(*			
	RafalOS
	Rafał Osajda		10.11.2025		TC 4024.66
	Główny blok konfiguracyjny MachineControl
*)
FUNCTION_BLOCK FB_MachineConfiguration EXTENDS FB_Base IMPLEMENTS ITF_MCConfiguration
VAR

END_VAR

(*			
	RafalOS
	Rafał Osajda		13.11.2025		TC 4024.66
	Metoda przeznaczona do dodawania elementów do FB_MachineControl
*)
METHOD AddElements : BOOL
VAR_INPUT
	itfMachineControl	: B_MachineControl.ITF_MCMachineControlConfigure;
END_VAR
END_METHOD

(*
	RafalOS
	Rafał Osajda		13.11.2025		TC 4024.66
	Dodanie samego siebie do systemu controli maszyny
*)
METHOD AddMachineCotrolToYourSelf : BOOL
VAR_INPUT
	itfMachineControl	: B_MachineControl.ITF_MCMachineControlConfigure;
END_VAR
END_METHOD

(*
	RafalOS
	Rafał Osajda		13.11.2025		TC 4024.66
	Dodanie modułu sterowania stanami i trybami do machinecontrol
*)
METHOD AddSaMCotrollerToMachineControl : BOOL
VAR_INPUT
	itfMachineControl	: B_MachineControl.ITF_MCMachineControlConfigure;
END_VAR
END_METHOD

(*			
	RafalOS
	Rafał Osajda		13.11.2025		TC 4024.66
	Zlinkowanie danych wspólnych do dodanych elementów
*)
METHOD LinkCommonDataToAddedElements : BOOL
VAR_INPUT
	itfMachineControl	: B_MachineControl.ITF_MCMachineControlConfigure;
END_VAR
END_METHOD

(*			
	RafalOS
	Rafał Osajda		13.11.2025		TC 4024.66
	Dodanie głównego komunikatora pomiędzy topelementami do topelementów
*)
METHOD LinkMassangerToaddedTopElements : BOOL
VAR_INPUT
	itfMachineControl	: B_MachineControl.ITF_MCMachineControlConfigure;
END_VAR
END_METHOD

(*			
	RafalOS
	Rafał Osajda		13.11.2025		TC 4024.66
	Podłączenie wsyzstkich zmiennych pochodzących od Programu safety 
*)
METHOD LinkSafetyToaddedElements : BOOL
VAR_INPUT
	itfMachineControl	: B_MachineControl.ITF_MCMachineControlConfigure;
END_VAR
END_METHOD

(*			
	RafalOS
	Rafał Osajda		13.11.2025		TC 4024.66
	Nadanie unikalnych kodów elementom w systemie
*)
METHOD SetCodeToAddedElements : BOOL
VAR_INPUT
	itfMachineControl	: B_MachineControl.ITF_MCMachineControlConfigure;
END_VAR
END_METHOD

(*			
	RafalOS
	Rafał Osajda		13.11.2025		TC 4024.66
	Nadaje unikalne ID zgłoszeniom dodanym do elementów w sesyemie
*)
METHOD SetIDEventsToAddedElements : BOOL
VAR_INPUT
	itfMachineControl	: B_MachineControl.ITF_MCMachineControlConfigure;
END_VAR
END_METHOD

(*			
	RafalOS
	Rafał Osajda		13.11.2025		TC 4024.66
	Dodanie wszystkim elementom w systemie unikalnego ID
*)
METHOD SetIDToAddedElements : BOOL
VAR_INPUT
	itfMachineControl	: B_MachineControl.ITF_MCMachineControlConfigure;
END_VAR
END_METHOD

END_FUNCTION_BLOCK

(* stored: Version 1.1.0.1, ProductVersion 3.1.4024.15
   POU FB_MachineConfiguration: Id {ee925a5b-f7fe-416e-8a33-e493e5327aae}, SpecialFunc None
   Method AddElements: Id {7b730765-41af-4c9b-9f6a-4c5a645abba8}
   Method AddMachineCotrolToYourSelf: Id {c8ed0d9d-f48c-476a-915b-a4eba002124b}
   Method AddSaMCotrollerToMachineControl: Id {01e4bd98-cea4-48b9-bac4-c2658d2eb279}
   Method LinkCommonDataToAddedElements: Id {ac0aabe4-15a4-490d-b3a0-5896b9031d05}
   Method LinkMassangerToaddedTopElements: Id {b7ca5c08-4047-434f-be66-47086ad067ba}
   Method LinkSafetyToaddedElements: Id {a7fb546a-9043-48d0-a215-0be12580516a}
   Method SetCodeToAddedElements: Id {10c39845-1161-4a70-8150-cbc008075584}
   Method SetIDEventsToAddedElements: Id {d886dcd7-8305-494f-9ced-3ff0d8f83511}
   Method SetIDToAddedElements: Id {3f3df8aa-f4cd-41e5-9f39-ff6b258bd4d3} *)
